// TwinCAT 3 PLC project SolidAttenuatorPLC
// ProgramVersion: 3.1.4022.7
// libraries:
//   lcls-twincat-motion, * (SLAC)
//   Tc2_Standard, * (Beckhoff Automation GmbH)
//   Tc2_System, * (Beckhoff Automation GmbH)
//   Tc3_Module, * (Beckhoff Automation GmbH)
//   VisuDialogs, * (System)
//   LCLS General,0.0.0,SLAC
//   VisuSymbols,3.5.10.0,System
// project tree:
//   DUTs/ DUT_MotionStage_Extras.TcDUT, ENUM_SXR_SATT_Position.TcDUT
//   / GlobalTextList.TcGTLO, PlcTask.TcTTO, VISU_TASK.TcTTO
//   GVLs/ Main.TcGVL
//   POUs/ FB_SXR_SATT_PositionState.TcPOU, FB_SXR_SATT_Stage.TcPOU, PRG_1_PlcTask.TcPOU, PRG_2_AT1K4.TcPOU
//   VISUs/ AT2K2_4022.TcVIS, VisualizationManager.TcVMO (not stored), VISU_MotionStage_4022.TcVIS, VISU_RTDs_4022.TcVIS
// real-time tasks:
//   TASK PlcTask: cycle T#10ms, priority 20, ADS port 350
//   TASK VISU_TASK: cycle T#200000us, priority 30, ADS port 351
// motion (NC):
//   TASK NC-Task 1 SAF: cycle T#2ms, priority 4, ADS port 501
//   TASK NC-Task 1 SVB: cycle T#10ms, priority 8, ADS port 511
//   AXIS AT1K4-M1 (id 1)
//     Dynamic: AccelerationMaximum=400, DecelerationMaximum=400, Acceleration=160, Deceleration=160, Jerk=80, DelayTime=0.008
//     Velo: Maximum=80
//     OtherSettings: AllowMotionCmdToSlave=true
//     encoder EncType=29
//       EncPara: ScaleFactorNumerator=5e-05, MaxCount=#xffffffff
//         SoftEndMinControl: Enable=true, Range=16.5
//         SoftEndMaxControl: Enable=true, Range=152.5
//         Inc: RefSoftSyncMask=#x0000ffff
//     drive DrvType=24
//       Analog: VeloReferenz=40, ScaleFactorActTorque=0.1
//       TimeComp: TaskDelayCycles=1
//     controller CtrType=2
//       CtrPara: PriorControlFactor=1
//         PosDiffControl: Range=0.2
//         PID: PosKp=20, PosExtKp=1, PosExtVelo=0.1
//         Observer: BandWidth=20
//   AXIS AT1K4-M2 (id 2)
//     Dynamic: AccelerationMaximum=400, DecelerationMaximum=400, Acceleration=160, Deceleration=160, Jerk=80, DelayTime=0.008
//     Velo: Maximum=80
//     OtherSettings: AllowMotionCmdToSlave=true
//     encoder EncType=29
//       EncPara: ScaleFactorNumerator=5e-05, MaxCount=#xffffffff, ReferenceSystem=1
//         SoftEndMinControl: Enable=true, Range=16.5
//         SoftEndMaxControl: Enable=true, Range=152.5
//         Inc: RefSoftSyncMask=#x0000ffff
//     drive DrvType=24
//       Analog: VeloReferenz=40, ScaleFactorActTorque=0.1
//       TimeComp: TaskDelayCycles=1
//     controller CtrType=2
//       CtrPara: PriorControlFactor=1
//         PosDiffControl: Range=0.2
//         PID: PosKp=20, PosExtKp=1, PosExtVelo=0.1
//         Observer: BandWidth=20
//   AXIS AT1K4-M3 (id 3)
//     Dynamic: AccelerationMaximum=400, DecelerationMaximum=400, Acceleration=160, Deceleration=160, Jerk=80, DelayTime=0.008
//     Velo: Maximum=80
//     OtherSettings: AllowMotionCmdToSlave=true
//     encoder EncType=29
//       EncPara: ScaleFactorNumerator=5e-05, MaxCount=#xffffffff, ReferenceSystem=1
//         SoftEndMinControl: Enable=true, Range=16.5
//         SoftEndMaxControl: Enable=true, Range=152.5
//         Inc: RefSoftSyncMask=#x0000ffff
//     drive DrvType=24
//       Analog: VeloReferenz=40, ScaleFactorActTorque=0.1
//       TimeComp: TaskDelayCycles=1
//     controller CtrType=2
//       CtrPara: PriorControlFactor=1
//         PosDiffControl: Range=0.2
//         PID: PosKp=20, PosExtKp=1, PosExtVelo=0.1
//         Observer: BandWidth=20
//   AXIS AT1K4-M4 (id 4)
//     Dynamic: AccelerationMaximum=400, DecelerationMaximum=400, Acceleration=160, Deceleration=160, Jerk=80, DelayTime=0.008
//     Velo: Maximum=80
//     OtherSettings: AllowMotionCmdToSlave=true
//     encoder EncType=29
//       EncPara: ScaleFactorNumerator=5e-05, MaxCount=#xffffffff, ReferenceSystem=1
//         SoftEndMinControl: Enable=true, Range=16.5
//         SoftEndMaxControl: Enable=true, Range=152.5
//         Inc: RefSoftSyncMask=#x0000ffff
//     drive DrvType=24
//       Analog: VeloReferenz=40, ScaleFactorActTorque=0.1
//       TimeComp: TaskDelayCycles=1
//     controller CtrType=2
//       CtrPara: PriorControlFactor=1
//         PosDiffControl: Range=0.2
//         PID: PosKp=20, PosExtKp=1, PosExtVelo=0.1
//         Observer: BandWidth=20
// I/O:
//   DEVICE Device 1 (EtherCAT), AmsNetId 172.21.148.185.2.1
//     Term 1 (EK1200) [EK1200-5000 EtherCAT Power supply (2A E-Bus)]
//       Term 14 (EL6695) [EL6695 EtherCAT Bridge terminal (Primary)]
//       Term 15 (EK1110) [EK1110 EtherCAT extension]
//     Term 16 (EK1100) [EK1100 EtherCAT Coupler (2A E-Bus)]
//       AT1K4-EL7047-01
//       AT1K4-EL7047-02 [EL7047 1Ch. Stepper motor output stage (50V, 5A)]
//       AT1K4-EL7047-03
//       AT1K4-EL7047-04
//       AT1K4-EL5042-01
//       AT1K4-EL5042-02
//       AT1K4-EL3202-01 [EL3202-0020 2Ch. Ana. Input PT100 (RTD), High Precision, calibrated]
//       AT1K4-EL3202-02 [EL3202-0020 2Ch. Ana. Input PT100 (RTD), High Precision, calibrated]
//       AT1K4-EL3202-03 [EL3202-0020 2Ch. Ana. Input PT100 (RTD), High Precision, calibrated]
//       AT1K4-EL3202-04 [EL3202-0020 2Ch. Ana. Input PT100 (RTD), High Precision, calibrated]
//       Term 12 (EL9011)
//   DEVICE Device 2 (EtherCAT Automation Protocol) (disabled), AmsNetId 172.21.148.185.3.1
//   DEVICE Device 5 (RT-Ethernet Protocol) (disabled), AmsNetId 172.21.148.185.6.1
//   DEVICE Device 4 (USB) (disabled)
//   DEVICE Device 6 (NOV-DP-RAM)
// variable links:
//   (this object) <-> Device 1 (EtherCAT)/Term 16 (EK1100)/AT1K4-EL5042-01
//     Enc/Inputs/In/nComState @bit 1 <-> WcState/InputToggle
//     Enc/Inputs/In/nComState <-> WcState/WcState
//     Enc/Inputs/In/nDataIn1 <-> FB Inputs Channel 1/Position
//     Enc/Inputs/In/nDataIn1 <-> FB Inputs Channel 2/Position
//     Enc/Inputs/In/nState1 @bit 12 <-> FB Inputs Channel 1/Status/Diag
//     Enc/Inputs/In/nState1 @bit 12 <-> FB Inputs Channel 2/Status/Diag
//     Enc/Inputs/In/nState1 @bit 1 <-> FB Inputs Channel 1/Status/Error
//     Enc/Inputs/In/nState1 @bit 1 <-> FB Inputs Channel 2/Status/Error
//     Enc/Inputs/In/nState1 @bit 14 <-> FB Inputs Channel 1/Status/Input cycle counter
//     Enc/Inputs/In/nState1 @bit 14 <-> FB Inputs Channel 2/Status/Input cycle counter
//     Enc/Inputs/In/nState1 @bit 2 <-> FB Inputs Channel 1/Status/Ready
//     Enc/Inputs/In/nState1 @bit 2 <-> FB Inputs Channel 2/Status/Ready
//     Enc/Inputs/In/nState1 @bit 13 <-> FB Inputs Channel 1/Status/TxPDO State
//     Enc/Inputs/In/nState1 @bit 13 <-> FB Inputs Channel 2/Status/TxPDO State
//     Enc/Inputs/In/nState1 <-> FB Inputs Channel 1/Status/Warning
//     Enc/Inputs/In/nState1 <-> FB Inputs Channel 2/Status/Warning
//   (this object) <-> Device 1 (EtherCAT)/Term 16 (EK1100)/AT1K4-EL7047-01
//     Drive/Inputs/In/nState1 @bit 3 <-> STM Status/Status/Error
//     Drive/Inputs/In/nState1 @bit 7 <-> STM Status/Status/Motor stall
//     Drive/Inputs/In/nState1 @bit 5 <-> STM Status/Status/Moving negative
//     Drive/Inputs/In/nState1 @bit 4 <-> STM Status/Status/Moving positive
//     Drive/Inputs/In/nState1 @bit 1 <-> STM Status/Status/Ready
//     Drive/Inputs/In/nState1 <-> STM Status/Status/Ready to enable
//     Drive/Inputs/In/nState1 @bit 6 <-> STM Status/Status/Torque reduced
//     Drive/Inputs/In/nState1 @bit 2 <-> STM Status/Status/Warning
//     Drive/Inputs/In/nState2 @bit 3 <-> STM Status/Status/Digital input 1
//     Drive/Inputs/In/nState2 @bit 4 <-> STM Status/Status/Digital input 2
//     Drive/Inputs/In/nState2 @bit 5 <-> STM Status/Status/Sync error
//     Drive/Inputs/In/nState2 @bit 7 <-> STM Status/Status/TxPDO Toggle
//     Drive/Inputs/In/nState4 @bit 1 <-> WcState/InputToggle
//     Drive/Inputs/In/nState4 <-> WcState/WcState
//     Drive/Outputs/Out/nCtrl1 <-> STM Control/Control/Enable
//     Drive/Outputs/Out/nCtrl1 @bit 2 <-> STM Control/Control/Reduce torque
//     Drive/Outputs/Out/nCtrl1 @bit 1 <-> STM Control/Control/Reset
//     Drive/Outputs/Out/nCtrl2 @bit 3 <-> STM Control/Control/Digital output 1
//     Drive/Outputs/Out/nDataOut2[0] <-> STM Velocity/Velocity
//   (this object) <-> Device 1 (EtherCAT)/Term 16 (EK1100)/AT1K4-EL7047-02
//     Drive/Inputs/In/nState1 @bit 3 <-> STM Status/Status/Error
//     Drive/Inputs/In/nState1 @bit 7 <-> STM Status/Status/Motor stall
//     Drive/Inputs/In/nState1 @bit 5 <-> STM Status/Status/Moving negative
//     Drive/Inputs/In/nState1 @bit 4 <-> STM Status/Status/Moving positive
//     Drive/Inputs/In/nState1 @bit 1 <-> STM Status/Status/Ready
//     Drive/Inputs/In/nState1 <-> STM Status/Status/Ready to enable
//     Drive/Inputs/In/nState1 @bit 6 <-> STM Status/Status/Torque reduced
//     Drive/Inputs/In/nState1 @bit 2 <-> STM Status/Status/Warning
//     Drive/Inputs/In/nState2 @bit 3 <-> STM Status/Status/Digital input 1
//     Drive/Inputs/In/nState2 @bit 4 <-> STM Status/Status/Digital input 2
//     Drive/Inputs/In/nState2 @bit 5 <-> STM Status/Status/Sync error
//     Drive/Inputs/In/nState2 @bit 7 <-> STM Status/Status/TxPDO Toggle
//     Drive/Inputs/In/nState4 @bit 1 <-> WcState/InputToggle
//     Drive/Inputs/In/nState4 <-> WcState/WcState
//     Drive/Outputs/Out/nCtrl1 <-> STM Control/Control/Enable
//     Drive/Outputs/Out/nCtrl1 @bit 2 <-> STM Control/Control/Reduce torque
//     Drive/Outputs/Out/nCtrl1 @bit 1 <-> STM Control/Control/Reset
//     Drive/Outputs/Out/nCtrl2 @bit 3 <-> STM Control/Control/Digital output 1
//     Drive/Outputs/Out/nDataOut2[0] <-> STM Velocity/Velocity
//   (this object) <-> Device 1 (EtherCAT)/Term 16 (EK1100)/AT1K4-EL5042-02
//     Enc/Inputs/In/nComState @bit 1 <-> WcState/InputToggle
//     Enc/Inputs/In/nComState <-> WcState/WcState
//     Enc/Inputs/In/nDataIn1 <-> FB Inputs Channel 1/Position
//     Enc/Inputs/In/nDataIn1 <-> FB Inputs Channel 2/Position
//     Enc/Inputs/In/nState1 @bit 12 <-> FB Inputs Channel 1/Status/Diag
//     Enc/Inputs/In/nState1 @bit 12 <-> FB Inputs Channel 2/Status/Diag
//     Enc/Inputs/In/nState1 @bit 1 <-> FB Inputs Channel 1/Status/Error
//     Enc/Inputs/In/nState1 @bit 1 <-> FB Inputs Channel 2/Status/Error
//     Enc/Inputs/In/nState1 @bit 14 <-> FB Inputs Channel 1/Status/Input cycle counter
//     Enc/Inputs/In/nState1 @bit 14 <-> FB Inputs Channel 2/Status/Input cycle counter
//     Enc/Inputs/In/nState1 @bit 2 <-> FB Inputs Channel 1/Status/Ready
//     Enc/Inputs/In/nState1 @bit 2 <-> FB Inputs Channel 2/Status/Ready
//     Enc/Inputs/In/nState1 @bit 13 <-> FB Inputs Channel 1/Status/TxPDO State
//     Enc/Inputs/In/nState1 @bit 13 <-> FB Inputs Channel 2/Status/TxPDO State
//     Enc/Inputs/In/nState1 <-> FB Inputs Channel 1/Status/Warning
//     Enc/Inputs/In/nState1 <-> FB Inputs Channel 2/Status/Warning
//   (this object) <-> Device 1 (EtherCAT)/Term 16 (EK1100)/AT1K4-EL7047-03
//     Drive/Inputs/In/nState1 @bit 3 <-> STM Status/Status/Error
//     Drive/Inputs/In/nState1 @bit 7 <-> STM Status/Status/Motor stall
//     Drive/Inputs/In/nState1 @bit 5 <-> STM Status/Status/Moving negative
//     Drive/Inputs/In/nState1 @bit 4 <-> STM Status/Status/Moving positive
//     Drive/Inputs/In/nState1 @bit 1 <-> STM Status/Status/Ready
//     Drive/Inputs/In/nState1 <-> STM Status/Status/Ready to enable
//     Drive/Inputs/In/nState1 @bit 6 <-> STM Status/Status/Torque reduced
//     Drive/Inputs/In/nState1 @bit 2 <-> STM Status/Status/Warning
//     Drive/Inputs/In/nState2 @bit 3 <-> STM Status/Status/Digital input 1
//     Drive/Inputs/In/nState2 @bit 4 <-> STM Status/Status/Digital input 2
//     Drive/Inputs/In/nState2 @bit 5 <-> STM Status/Status/Sync error
//     Drive/Inputs/In/nState2 @bit 7 <-> STM Status/Status/TxPDO Toggle
//     Drive/Inputs/In/nState4 @bit 1 <-> WcState/InputToggle
//     Drive/Inputs/In/nState4 <-> WcState/WcState
//     Drive/Outputs/Out/nCtrl1 <-> STM Control/Control/Enable
//     Drive/Outputs/Out/nCtrl1 @bit 2 <-> STM Control/Control/Reduce torque
//     Drive/Outputs/Out/nCtrl1 @bit 1 <-> STM Control/Control/Reset
//     Drive/Outputs/Out/nCtrl2 @bit 3 <-> STM Control/Control/Digital output 1
//     Drive/Outputs/Out/nDataOut2[0] <-> STM Velocity/Velocity
//   (this object) <-> Device 1 (EtherCAT)/Term 16 (EK1100)/AT1K4-EL7047-04
//     Drive/Inputs/In/nState1 @bit 3 <-> STM Status/Status/Error
//     Drive/Inputs/In/nState1 @bit 7 <-> STM Status/Status/Motor stall
//     Drive/Inputs/In/nState1 @bit 5 <-> STM Status/Status/Moving negative
//     Drive/Inputs/In/nState1 @bit 4 <-> STM Status/Status/Moving positive
//     Drive/Inputs/In/nState1 @bit 1 <-> STM Status/Status/Ready
//     Drive/Inputs/In/nState1 <-> STM Status/Status/Ready to enable
//     Drive/Inputs/In/nState1 @bit 6 <-> STM Status/Status/Torque reduced
//     Drive/Inputs/In/nState1 @bit 2 <-> STM Status/Status/Warning
//     Drive/Inputs/In/nState2 @bit 3 <-> STM Status/Status/Digital input 1
//     Drive/Inputs/In/nState2 @bit 4 <-> STM Status/Status/Digital input 2
//     Drive/Inputs/In/nState2 @bit 5 <-> STM Status/Status/Sync error
//     Drive/Inputs/In/nState2 @bit 7 <-> STM Status/Status/TxPDO Toggle
//     Drive/Inputs/In/nState4 @bit 1 <-> WcState/InputToggle
//     Drive/Inputs/In/nState4 <-> WcState/WcState
//     Drive/Outputs/Out/nCtrl1 <-> STM Control/Control/Enable
//     Drive/Outputs/Out/nCtrl1 @bit 2 <-> STM Control/Control/Reduce torque
//     Drive/Outputs/Out/nCtrl1 @bit 1 <-> STM Control/Control/Reset
//     Drive/Outputs/Out/nCtrl2 @bit 3 <-> STM Control/Control/Digital output 1
//     Drive/Outputs/Out/nDataOut2[0] <-> STM Velocity/Velocity
//   SolidAttenuatorPLC Instance <-> Device 1 (EtherCAT)/Term 16 (EK1100)/AT1K4-EL3202-01
//     PlcTask Inputs/PRG_2_AT1K4.fbStage1.fbRTD_1.bError <-> RTD Inputs Channel 1/Status/Error
//     PlcTask Inputs/PRG_2_AT1K4.fbStage1.fbRTD_2.bError <-> RTD Inputs Channel 2/Status/Error
//     PlcTask Inputs/PRG_2_AT1K4.fbStage1.fbRTD_1.bOverrange <-> RTD Inputs Channel 1/Status/Overrange
//     PlcTask Inputs/PRG_2_AT1K4.fbStage1.fbRTD_2.bOverrange <-> RTD Inputs Channel 2/Status/Overrange
//     PlcTask Inputs/PRG_2_AT1K4.fbStage1.fbRTD_1.bUnderrange <-> RTD Inputs Channel 1/Status/Underrange
//     PlcTask Inputs/PRG_2_AT1K4.fbStage1.fbRTD_2.bUnderrange <-> RTD Inputs Channel 2/Status/Underrange
//     PlcTask Inputs/PRG_2_AT1K4.fbStage1.fbRTD_1.iRaw <-> RTD Inputs Channel 1/Value
//     PlcTask Inputs/PRG_2_AT1K4.fbStage1.fbRTD_2.iRaw <-> RTD Inputs Channel 2/Value
//   SolidAttenuatorPLC Instance <-> Device 1 (EtherCAT)/Term 16 (EK1100)/AT1K4-EL3202-02
//     PlcTask Inputs/PRG_2_AT1K4.fbStage2.fbRTD_1.bError <-> RTD Inputs Channel 1/Status/Error
//     PlcTask Inputs/PRG_2_AT1K4.fbStage2.fbRTD_2.bError <-> RTD Inputs Channel 2/Status/Error
//     PlcTask Inputs/PRG_2_AT1K4.fbStage2.fbRTD_1.bOverrange <-> RTD Inputs Channel 1/Status/Overrange
//     PlcTask Inputs/PRG_2_AT1K4.fbStage2.fbRTD_2.bOverrange <-> RTD Inputs Channel 2/Status/Overrange
//     PlcTask Inputs/PRG_2_AT1K4.fbStage2.fbRTD_1.bUnderrange <-> RTD Inputs Channel 1/Status/Underrange
//     PlcTask Inputs/PRG_2_AT1K4.fbStage2.fbRTD_2.bUnderrange <-> RTD Inputs Channel 2/Status/Underrange
//     PlcTask Inputs/PRG_2_AT1K4.fbStage2.fbRTD_1.iRaw <-> RTD Inputs Channel 1/Value
//     PlcTask Inputs/PRG_2_AT1K4.fbStage2.fbRTD_2.iRaw <-> RTD Inputs Channel 2/Value
//   SolidAttenuatorPLC Instance <-> Device 1 (EtherCAT)/Term 16 (EK1100)/AT1K4-EL3202-03
//     PlcTask Inputs/PRG_2_AT1K4.fbStage3.fbRTD_1.bError <-> RTD Inputs Channel 1/Status/Error
//     PlcTask Inputs/PRG_2_AT1K4.fbStage3.fbRTD_2.bError <-> RTD Inputs Channel 2/Status/Error
//     PlcTask Inputs/PRG_2_AT1K4.fbStage3.fbRTD_1.bOverrange <-> RTD Inputs Channel 1/Status/Overrange
//     PlcTask Inputs/PRG_2_AT1K4.fbStage3.fbRTD_2.bOverrange <-> RTD Inputs Channel 2/Status/Overrange
//     PlcTask Inputs/PRG_2_AT1K4.fbStage3.fbRTD_1.bUnderrange <-> RTD Inputs Channel 1/Status/Underrange
//     PlcTask Inputs/PRG_2_AT1K4.fbStage3.fbRTD_2.bUnderrange <-> RTD Inputs Channel 2/Status/Underrange
//     PlcTask Inputs/PRG_2_AT1K4.fbStage3.fbRTD_1.iRaw <-> RTD Inputs Channel 1/Value
//     PlcTask Inputs/PRG_2_AT1K4.fbStage3.fbRTD_2.iRaw <-> RTD Inputs Channel 2/Value
//   SolidAttenuatorPLC Instance <-> Device 1 (EtherCAT)/Term 16 (EK1100)/AT1K4-EL3202-04
//     PlcTask Inputs/PRG_2_AT1K4.fbStage4.fbRTD_1.bError <-> RTD Inputs Channel 1/Status/Error
//     PlcTask Inputs/PRG_2_AT1K4.fbStage4.fbRTD_2.bError <-> RTD Inputs Channel 2/Status/Error
//     PlcTask Inputs/PRG_2_AT1K4.fbStage4.fbRTD_1.bOverrange <-> RTD Inputs Channel 1/Status/Overrange
//     PlcTask Inputs/PRG_2_AT1K4.fbStage4.fbRTD_2.bOverrange <-> RTD Inputs Channel 2/Status/Overrange
//     PlcTask Inputs/PRG_2_AT1K4.fbStage4.fbRTD_1.bUnderrange <-> RTD Inputs Channel 1/Status/Underrange
//     PlcTask Inputs/PRG_2_AT1K4.fbStage4.fbRTD_2.bUnderrange <-> RTD Inputs Channel 2/Status/Underrange
//     PlcTask Inputs/PRG_2_AT1K4.fbStage4.fbRTD_1.iRaw <-> RTD Inputs Channel 1/Value
//     PlcTask Inputs/PRG_2_AT1K4.fbStage4.fbRTD_2.iRaw <-> RTD Inputs Channel 2/Value
//   SolidAttenuatorPLC Instance <-> Device 1 (EtherCAT)/Term 16 (EK1100)/AT1K4-EL5042-01
//     PlcTask Inputs/Main.M1.nRawEncoderULINT <-> FB Inputs Channel 1/Position
//     PlcTask Inputs/Main.M2.nRawEncoderULINT <-> FB Inputs Channel 2/Position
//   SolidAttenuatorPLC Instance <-> Device 1 (EtherCAT)/Term 16 (EK1100)/AT1K4-EL5042-02
//     PlcTask Inputs/Main.M3.nRawEncoderULINT <-> FB Inputs Channel 1/Position
//     PlcTask Inputs/Main.M4.nRawEncoderULINT <-> FB Inputs Channel 2/Position
//   SolidAttenuatorPLC Instance <-> Device 1 (EtherCAT)/Term 16 (EK1100)/AT1K4-EL7047-01
//     PlcTask Inputs/Main.M1.bLimitBackwardEnable <-> STM Status/Status/Digital input 2
//     PlcTask Inputs/Main.M1.bLimitForwardEnable <-> STM Status/Status/Digital input 1
//   SolidAttenuatorPLC Instance <-> Device 1 (EtherCAT)/Term 16 (EK1100)/AT1K4-EL7047-02
//     PlcTask Inputs/Main.M2.bLimitBackwardEnable <-> STM Status/Status/Digital input 2
//     PlcTask Inputs/Main.M2.bLimitForwardEnable <-> STM Status/Status/Digital input 1
//   SolidAttenuatorPLC Instance <-> Device 1 (EtherCAT)/Term 16 (EK1100)/AT1K4-EL7047-03
//     PlcTask Inputs/Main.M3.bLimitBackwardEnable <-> STM Status/Status/Digital input 2
//     PlcTask Inputs/Main.M3.bLimitForwardEnable <-> STM Status/Status/Digital input 1
//   SolidAttenuatorPLC Instance <-> Device 1 (EtherCAT)/Term 16 (EK1100)/AT1K4-EL7047-04
//     PlcTask Inputs/Main.M4.bLimitBackwardEnable <-> STM Status/Status/Digital input 2
//     PlcTask Inputs/Main.M4.bLimitForwardEnable <-> STM Status/Status/Digital input 1
//   SolidAttenuatorPLC Instance <-> NC-Task 1 SAF/Axes/AT1K4-M1
//     PlcTask Inputs/Main.M1.Axis.NcToPlc <-> Outputs/ToPlc
//     PlcTask Outputs/Main.M1.Axis.PlcToNc <-> Inputs/FromPlc
//   SolidAttenuatorPLC Instance <-> NC-Task 1 SAF/Axes/AT1K4-M2
//     PlcTask Inputs/Main.M2.Axis.NcToPlc <-> Outputs/ToPlc
//     PlcTask Outputs/Main.M2.Axis.PlcToNc <-> Inputs/FromPlc
//   SolidAttenuatorPLC Instance <-> NC-Task 1 SAF/Axes/AT1K4-M3
//     PlcTask Inputs/Main.M3.Axis.NcToPlc <-> Outputs/ToPlc
//     PlcTask Outputs/Main.M3.Axis.PlcToNc <-> Inputs/FromPlc
//   SolidAttenuatorPLC Instance <-> NC-Task 1 SAF/Axes/AT1K4-M4
//     PlcTask Inputs/Main.M4.Axis.NcToPlc <-> Outputs/ToPlc
//     PlcTask Outputs/Main.M4.Axis.PlcToNc <-> Inputs/FromPlc

CONFIGURATION SolidAttenuatorPLC
    RESOURCE PLC ON TwinCAT3
        TASK PlcTask(INTERVAL := T#10ms, PRIORITY := 20);
        TASK VISU_TASK(INTERVAL := T#200000us, PRIORITY := 30);
        PROGRAM PRG_1_PlcTask WITH PlcTask : PRG_1_PlcTask;
        PROGRAM VisuElems_Visu_Prg WITH VISU_TASK : VisuElems.Visu_Prg;
    END_RESOURCE
END_CONFIGURATION

// ---- DUTs/DUT_MotionStage_Extras.TcDUT
TYPE DUT_MotionStage_Extras :
STRUCT
    fVisuStep: LREAL;
    bVisuLowLim: BOOL;
    bVisuHighLim: BOOL;
END_STRUCT
END_TYPE

// ---- DUTs/ENUM_SXR_SATT_Position.TcDUT
{attribute 'qualified_only'}
TYPE ENUM_SXR_SATT_Position :
(
    UNKNOWN := 0, // UNKNOWN must be in slot 0 or the FB breaks
    OUT := 1, // OUT at slot 1 is a convention
    FILTER1 := 2,
    FILTER2 := 3,
    FILTER3 := 4,
    FILTER4 := 5
);
END_TYPE

// ---- GVLs/Main.TcGVL
{attribute 'qualified_only'}
VAR_GLOBAL
(*
    Only includes motor definitions for the IOC
    These are hard-coded to be Main.M#,
    but are very convenient to store in a GVL,
    hence the confusing namespace here

    This should be refactored once the IOC
    supports arbitrary ads paths for motors
*)
(*
    Four identical systems:
    Instr.		Area		ID#			Z (m)
    TMO			FEE			AT1K4-SOLID	748
    NEH 2.2		H2.2		AT1K2-SOLID	784
    NEH 2.2		H2.2		AT2K2-SOLID	788.8
    TXI			H1.1		AT1K3-SOLID	~763

*)
    {attribute 'pytmc' := 'pv: AT1K4:L2SI:MMS:01'}
    {attribute 'TcLinkTo' := '
        .bLimitForwardEnable  := TIIB[AT1K4-EL7047-01]^STM Status^Status^Digital input 1;
        .bLimitBackwardEnable := TIIB[AT1K4-EL7047-01]^STM Status^Status^Digital input 2;
        .nRawEncoderULINT     := TIIB[AT1K4-EL5042-01]^FB Inputs Channel 1^Position;
    '}
    M1: DUT_MotionStage := (sName := 'AT1K4:L2SI:MMS:01');

    {attribute 'pytmc' := 'pv: AT1K4:L2SI:MMS:02'}
    {attribute 'TcLinkTo' := '
        .bLimitForwardEnable  := TIIB[AT1K4-EL7047-02]^STM Status^Status^Digital input 1;
        .bLimitBackwardEnable := TIIB[AT1K4-EL7047-02]^STM Status^Status^Digital input 2;
        .nRawEncoderULINT     := TIIB[AT1K4-EL5042-01]^FB Inputs Channel 2^Position;
    '}
    M2: DUT_MotionStage := (sName := 'AT1K4:L2SI:MMS:02');

    {attribute 'pytmc' := 'pv: AT1K4:L2SI:MMS:03'}
    {attribute 'TcLinkTo' := '
        .bLimitForwardEnable  := TIIB[AT1K4-EL7047-03]^STM Status^Status^Digital input 1;
        .bLimitBackwardEnable := TIIB[AT1K4-EL7047-03]^STM Status^Status^Digital input 2;
        .nRawEncoderULINT     := TIIB[AT1K4-EL5042-02]^FB Inputs Channel 1^Position;
    '}
    M3: DUT_MotionStage := (sName := 'AT1K4:L2SI:MMS:03');

    {attribute 'pytmc' := 'pv: AT1K4:L2SI:MMS:04'}
    {attribute 'TcLinkTo' := '
        .bLimitForwardEnable  := TIIB[AT1K4-EL7047-04]^STM Status^Status^Digital input 1;
        .bLimitBackwardEnable := TIIB[AT1K4-EL7047-04]^STM Status^Status^Digital input 2;
        .nRawEncoderULINT     := TIIB[AT1K4-EL5042-02]^FB Inputs Channel 2^Position;
    '}
    M4: DUT_MotionStage := (sName := 'AT1K4:L2SI:MMS:04');

END_VAR

// ---- POUs/PRG_1_PlcTask.TcPOU

PROGRAM PRG_1_PlcTask
VAR
    fbLogHandler: FB_LogHandler;
END_VAR

fbLogHandler();

PRG_2_AT1K4();

END_PROGRAM

// ---- POUs/PRG_2_AT1K4.TcPOU
PROGRAM PRG_2_AT1K4
VAR
    (* TODO: use FALSE for simulation and production *)
    (* TODO: use TRUE when relying on visualization + actual hardware *)
    bDebug : BOOL := FALSE;

    nEnableMode : ENUM_StageEnableMode;

    {attribute 'pytmc' := 'pv: AT1K4:L2SI:MMS:01'}
    {attribute 'TcLinkTo' := '

        .fbRTD_1.iRaw := TIIB[AT1K4-EL3202-01]^RTD Inputs Channel 1^Value;
        .fbRTD_1.bError := TIIB[AT1K4-EL3202-01]^RTD Inputs Channel 1^Status^Error;
        .fbRTD_1.bUnderrange := TIIB[AT1K4-EL3202-01]^RTD Inputs Channel 1^Status^Underrange;
        .fbRTD_1.bOverrange := TIIB[AT1K4-EL3202-01]^RTD Inputs Channel 1^Status^Overrange;

        .fbRTD_2.iRaw := TIIB[AT1K4-EL3202-01]^RTD Inputs Channel 2^Value;
        .fbRTD_2.bError := TIIB[AT1K4-EL3202-01]^RTD Inputs Channel 2^Status^Error;
        .fbRTD_2.bUnderrange := TIIB[AT1K4-EL3202-01]^RTD Inputs Channel 2^Status^Underrange;
        .fbRTD_2.bOverrange := TIIB[AT1K4-EL3202-01]^RTD Inputs Channel 2^Status^Overrange;

    '}
    fbStage1: FB_SXR_SATT_Stage;

    {attribute 'pytmc' := 'pv: AT1K4:L2SI:MMS:02'}
    {attribute 'TcLinkTo' := '

        .fbRTD_1.iRaw := TIIB[AT1K4-EL3202-02]^RTD Inputs Channel 1^Value;
        .fbRTD_1.bError := TIIB[AT1K4-EL3202-02]^RTD Inputs Channel 1^Status^Error;
        .fbRTD_1.bUnderrange := TIIB[AT1K4-EL3202-02]^RTD Inputs Channel 1^Status^Underrange;
        .fbRTD_1.bOverrange := TIIB[AT1K4-EL3202-02]^RTD Inputs Channel 1^Status^Overrange;

        .fbRTD_2.iRaw := TIIB[AT1K4-EL3202-02]^RTD Inputs Channel 2^Value;
        .fbRTD_2.bError := TIIB[AT1K4-EL3202-02]^RTD Inputs Channel 2^Status^Error;
        .fbRTD_2.bUnderrange := TIIB[AT1K4-EL3202-02]^RTD Inputs Channel 2^Status^Underrange;
        .fbRTD_2.bOverrange := TIIB[AT1K4-EL3202-02]^RTD Inputs Channel 2^Status^Overrange;

    '}
    fbStage2: FB_SXR_SATT_Stage;

    {attribute 'pytmc' := 'pv: AT1K4:L2SI:MMS:03'}
    {attribute 'TcLinkTo' := '

        .fbRTD_1.iRaw := TIIB[AT1K4-EL3202-03]^RTD Inputs Channel 1^Value;
        .fbRTD_1.bError := TIIB[AT1K4-EL3202-03]^RTD Inputs Channel 1^Status^Error;
        .fbRTD_1.bUnderrange := TIIB[AT1K4-EL3202-03]^RTD Inputs Channel 1^Status^Underrange;
        .fbRTD_1.bOverrange := TIIB[AT1K4-EL3202-03]^RTD Inputs Channel 1^Status^Overrange;

        .fbRTD_2.iRaw := TIIB[AT1K4-EL3202-03]^RTD Inputs Channel 2^Value;
        .fbRTD_2.bError := TIIB[AT1K4-EL3202-03]^RTD Inputs Channel 2^Status^Error;
        .fbRTD_2.bUnderrange := TIIB[AT1K4-EL3202-03]^RTD Inputs Channel 2^Status^Underrange;
        .fbRTD_2.bOverrange := TIIB[AT1K4-EL3202-03]^RTD Inputs Channel 2^Status^Overrange;
    '}
    fbStage3: FB_SXR_SATT_Stage;

    {attribute 'pytmc' := 'pv: AT1K4:L2SI:MMS:04'}
    {attribute 'TcLinkTo' := '

        .fbRTD_1.iRaw := TIIB[AT1K4-EL3202-04]^RTD Inputs Channel 1^Value;
        .fbRTD_1.bError := TIIB[AT1K4-EL3202-04]^RTD Inputs Channel 1^Status^Error;
        .fbRTD_1.bUnderrange := TIIB[AT1K4-EL3202-04]^RTD Inputs Channel 1^Status^Underrange;
        .fbRTD_1.bOverrange := TIIB[AT1K4-EL3202-04]^RTD Inputs Channel 1^Status^Overrange;

        .fbRTD_2.iRaw := TIIB[AT1K4-EL3202-04]^RTD Inputs Channel 2^Value;
        .fbRTD_2.bError := TIIB[AT1K4-EL3202-04]^RTD Inputs Channel 2^Status^Error;
        .fbRTD_2.bUnderrange := TIIB[AT1K4-EL3202-04]^RTD Inputs Channel 2^Status^Underrange;
        .fbRTD_2.bOverrange := TIIB[AT1K4-EL3202-04]^RTD Inputs Channel 2^Status^Overrange;
    '}
    fbStage4: FB_SXR_SATT_Stage;

END_VAR

IF bDebug THEN
    // NEVER: checkouts with the TwinCAT NC GUI.
    nEnableMode := ENUM_StageEnableMode.NEVER;
ELSE
    // ALWAYS: want active position correction at all times
    nEnableMode := ENUM_StageEnableMode.ALWAYS;
END_IF

(* State setup - stage 1 *)
fbStage1.stOut.sName         := 'Out';
fbStage1.stOut.fPosition     := 50;
fbStage1.stOut.fDelta        := 100;
fbStage1.stOut.fVelocity     := 10;
fbStage1.stOut.bValid        := TRUE;
fbStage1.stOut.bMoveOk       := TRUE;

fbStage1.stFilter1.sName     := 'Filter 1';
fbStage1.stFilter1.fPosition := 500;
fbStage1.stFilter1.fDelta    := 0;
fbStage1.stFilter1.fVelocity := 10;
fbStage1.stFilter1.bValid    := FALSE;
fbStage1.stFilter1.bMoveOk   := FALSE;

fbStage1.stFilter2.sName     := 'Filter 2';
fbStage1.stFilter2.fPosition := 500;
fbStage1.stFilter2.fDelta    := 0;
fbStage1.stFilter2.fVelocity := 10;
fbStage1.stFilter2.bValid    := FALSE;
fbStage1.stFilter2.bMoveOk   := FALSE;

fbStage1.stFilter3.sName     := 'Filter 3';
fbStage1.stFilter3.fPosition := 500;
fbStage1.stFilter3.fDelta    := 0;
fbStage1.stFilter3.fVelocity := 10;
fbStage1.stFilter3.bValid    := FALSE;
fbStage1.stFilter3.bMoveOk   := FALSE;

fbStage1.stFilter4.sName     := 'Filter 4';
fbStage1.stFilter4.fPosition := 500;
fbStage1.stFilter4.fDelta    := 0;
fbStage1.stFilter4.fVelocity := 10;
fbStage1.stFilter4.bValid    := FALSE;
fbStage1.stFilter4.bMoveOk   := FALSE;

fbStage1(stAxis:=Main.M1, nEnableMode:=nEnableMode);

(* State setup - stage 2 *)
fbStage2.stOut.sName         := 'Out';
fbStage2.stOut.fPosition     := 50;
fbStage2.stOut.fDelta        := 100;
fbStage2.stOut.fVelocity     := 10;
fbStage2.stOut.bValid        := TRUE;
fbStage2.stOut.bMoveOk       := TRUE;

fbStage2.stFilter1.sName     := 'Filter 1';
fbStage2.stFilter1.fPosition := 500;
fbStage2.stFilter1.fDelta    := 0;
fbStage2.stFilter1.fVelocity := 10;
fbStage2.stFilter1.bValid    := FALSE;
fbStage2.stFilter1.bMoveOk   := FALSE;

fbStage2.stFilter2.sName     := 'Filter 2';
fbStage2.stFilter2.fPosition := 500;
fbStage2.stFilter2.fDelta    := 0;
fbStage2.stFilter2.fVelocity := 10;
fbStage2.stFilter2.bValid    := FALSE;
fbStage2.stFilter2.bMoveOk   := FALSE;

fbStage2.stFilter3.sName     := 'Filter 3';
fbStage2.stFilter3.fPosition := 500;
fbStage2.stFilter3.fDelta    := 0;
fbStage2.stFilter3.fVelocity := 10;
fbStage2.stFilter3.bValid    := FALSE;
fbStage2.stFilter3.bMoveOk   := FALSE;

fbStage2.stFilter4.sName     := 'Filter 4';
fbStage2.stFilter4.fPosition := 500;
fbStage2.stFilter4.fDelta    := 0;
fbStage2.stFilter4.fVelocity := 10;
fbStage2.stFilter4.bValid    := FALSE;
fbStage2.stFilter4.bMoveOk   := FALSE;

fbStage2(stAxis:=Main.M2, nEnableMode:=nEnableMode);

(* State setup - stage 3 *)
fbStage3.stOut.sName         := 'Out';
fbStage3.stOut.fPosition     := 50;
fbStage3.stOut.fDelta        := 100;
fbStage3.stOut.fVelocity     := 10;
fbStage3.stOut.bValid        := TRUE;
fbStage3.stOut.bMoveOk       := TRUE;

fbStage3.stFilter1.sName     := 'Filter 1';
fbStage3.stFilter1.fPosition := 500;
fbStage3.stFilter1.fDelta    := 0;
fbStage3.stFilter1.fVelocity := 10;
fbStage3.stFilter1.bValid    := FALSE;
fbStage3.stFilter1.bMoveOk   := FALSE;

fbStage3.stFilter2.sName     := 'Filter 2';
fbStage3.stFilter2.fPosition := 500;
fbStage3.stFilter2.fDelta    := 0;
fbStage3.stFilter2.fVelocity := 10;
fbStage3.stFilter2.bValid    := FALSE;
fbStage3.stFilter2.bMoveOk   := FALSE;

fbStage3.stFilter3.sName     := 'Filter 3';
fbStage3.stFilter3.fPosition := 500;
fbStage3.stFilter3.fDelta    := 0;
fbStage3.stFilter3.fVelocity := 10;
fbStage3.stFilter3.bValid    := FALSE;
fbStage3.stFilter3.bMoveOk   := FALSE;

fbStage3.stFilter4.sName     := 'Filter 4';
fbStage3.stFilter4.fPosition := 500;
fbStage3.stFilter4.fDelta    := 0;
fbStage3.stFilter4.fVelocity := 10;
fbStage3.stFilter4.bValid    := FALSE;
fbStage3.stFilter4.bMoveOk   := FALSE;

fbStage3(stAxis:=Main.M3, nEnableMode:=nEnableMode);

(* State setup - stage 4 *)
fbStage4.stOut.sName         := 'Out';
fbStage4.stOut.fPosition     := 50;
fbStage4.stOut.fDelta        := 100;
fbStage4.stOut.fVelocity     := 10;
fbStage4.stOut.bValid        := TRUE;
fbStage4.stOut.bMoveOk       := TRUE;

fbStage4.stFilter1.sName     := 'Filter 1';
fbStage4.stFilter1.fPosition := 500;
fbStage4.stFilter1.fDelta    := 0;
fbStage4.stFilter1.fVelocity := 10;
fbStage4.stFilter1.bValid    := FALSE;
fbStage4.stFilter1.bMoveOk   := FALSE;

fbStage4.stFilter2.sName     := 'Filter 2';
fbStage4.stFilter2.fPosition := 500;
fbStage4.stFilter2.fDelta    := 0;
fbStage4.stFilter2.fVelocity := 10;
fbStage4.stFilter2.bValid    := FALSE;
fbStage4.stFilter2.bMoveOk   := FALSE;

fbStage4.stFilter3.sName     := 'Filter 3';
fbStage4.stFilter3.fPosition := 500;
fbStage4.stFilter3.fDelta    := 0;
fbStage4.stFilter3.fVelocity := 10;
fbStage4.stFilter3.bValid    := FALSE;
fbStage4.stFilter3.bMoveOk   := FALSE;

fbStage4.stFilter4.sName     := 'Filter 4';
fbStage4.stFilter4.fPosition := 500;
fbStage4.stFilter4.fDelta    := 0;
fbStage4.stFilter4.fVelocity := 10;
fbStage4.stFilter4.bValid    := FALSE;
fbStage4.stFilter4.bMoveOk   := FALSE;

fbStage4(stAxis:=Main.M4, nEnableMode:=nEnableMode);

END_PROGRAM

// ---- POUs/FB_SXR_SATT_Stage.TcPOU
FUNCTION_BLOCK FB_SXR_SATT_Stage
VAR_IN_OUT
    stAxis : DUT_MotionStage;
END_VAR
VAR_INPUT
    nEnableMode : ENUM_StageEnableMode;

    stOut		: DUT_PositionState;
    stFilter1	: DUT_PositionState;
    stFilter2	: DUT_PositionState;
    stFilter3	: DUT_PositionState;
    stFilter4	: DUT_PositionState;
END_VAR
VAR_OUTPUT
    stExtra : DUT_MotionStage_Extras;
    fTemp1 : LREAL;
    fTemp2 : LREAL;
END_VAR
VAR
    // TODO: debug
    // fbMotion: FB_MotionStage;
    fbMotion: FB_MotionStageSim;

    {attribute 'pytmc' := '
         pv: STATE
    '}
    fbState 	: FB_SXR_SATT_PositionState;

    bInitialized: BOOL := FALSE;

    (* EL3202-0020: 0.01 °C per digit *)
    {attribute 'pytmc' := 'pv: RTD:1'}
    fbRTD_1: FB_TempSensor := ( fResolution:=0.01 );
    {attribute 'pytmc' := 'pv: RTD:2'}
    fbRTD_2: FB_TempSensor := ( fResolution:=0.01 );

END_VAR

IF NOT bInitialized THEN
    bInitialized := TRUE;

    (* Defaults for DUT_MotionStage *)
    stAxis.bHardwareEnable      := TRUE;
    stAxis.bLimitBackwardEnable := TRUE;
    stAxis.bLimitForwardEnable  := TRUE;
    stAxis.bPowerSelf           := TRUE;
    stAxis.nBrakeMode           := ENUM_StageBrakeMode.NO_BRAKE;
    stAxis.nHomingMode          := ENUM_EpicsHomeCmd.NONE;

    (* Defaults for visualization *)
    stExtra.fVisuStep			:= 0.1;

END_IF

fbRTD_1();
fTemp1 := fbRTD_1.fTemp;

fbRTD_2();
fTemp2 := fbRTD_2.fTemp;

stAxis.nEnableMode := nEnableMode;
fbMotion(stMotionStage:=stAxis);
fbState(
    bEnable:=TRUE,
    bReset:=FALSE,
    stMotionStage:=stAxis,
    stOut:=stOut,
    stFilter1:=stFilter1,
    stFilter2:=stFilter2,
    stFilter3:=stFilter3,
    stFilter4:=stFilter4
);

stExtra.bVisuHighLim := NOT stAxis.bAllForwardEnable;
stExtra.bVisuLowLim := NOT stAxis.bAllBackwardEnable;

END_FUNCTION_BLOCK

// ---- POUs/FB_SXR_SATT_PositionState.TcPOU
FUNCTION_BLOCK FB_SXR_SATT_PositionState EXTENDS FB_PositionStateBase
VAR_INPUT
     // The enum position to move to
     {attribute 'pytmc' := '
         pv: SET
         io: io
     '}
     enumSet: ENUM_SXR_SATT_Position;

    // NOTE: Do not pragma these, let it happen in the manager.
     // Information about the OUT position
     stOut		: DUT_PositionState;
     stFilter1	: DUT_PositionState;
     stFilter2	: DUT_PositionState;
     stFilter3	: DUT_PositionState;
     stFilter4	: DUT_PositionState;

END_VAR
VAR_OUTPUT
    // The enum state readback
    {attribute 'pytmc' := '
        pv: GET
        io: i
    '}
    enumGet: ENUM_SXR_SATT_Position;
END_VAR
VAR
    bInitialized: BOOL := FALSE;
END_VAR

IF NOT bInitialized THEN
    bInitialized := TRUE;

    arrStates[1] := stOut;
    arrStates[2] := stFilter1;
    arrStates[3] := stFilter2;
    arrStates[4] := stFilter3;
    arrStates[5] := stFilter4;

END_IF
setState := enumSet;
Exec();
enumGet := getState;
enumSet := setState;

END_FUNCTION_BLOCK

// ---- GlobalTextList.TcGTLO
TEXTLIST GlobalTextList
  468 = '%d'
  405 = '%f'
  425 = '%X'
  417 = '+'
  411 = '-'
  421 = '0 = Default Acceleration'
  423 = '0 = Default Deceleration'
  420 = 'Acceleration: %f'
  966 = 'Admin'
  17 = 'Axis 1'
  746 = 'Axis 2'
  124 = 'Axis 3'
  441 = 'Axis 4'
  650 = 'Axis X'
  588 = 'Channel 1: %.2f C'
  84 = 'Channel 1: %f C'
  809 = 'Channel 2: %.2f C'
  18 = 'Channel 2: %f C'
  415 = 'Clear'
  409 = 'Control'
  406 = 'Current Position'
  463 = 'Current Position (raw)'
  422 = 'Deceleration: %f'
  426 = 'Error Code'
  424 = 'Error:'
  413 = 'GO'
  414 = 'GO to set position'
  407 = 'High Limit Hit Indicator'
  404 = 'Low Limit Hit Indicator'
  408 = 'Moving:'
  823 = 'None'
  269 = 'Operator'
  721 = 'RTD1: %f C'
  433 = 'RTD2: %f C'
  878 = 'Service'
  410 = 'Set Position'
  418 = 'Settings'
  403 = 'Status'
  412 = 'Step Size'
  416 = 'STOP'
  917 = 'Temp 1: %f C'
  719 = 'Temp 2: %f C'
  647 = 'Temperature Sensors'
  865 = 'Thermocouple Readback'
  419 = 'Velocity: %f'
END_TEXTLIST

// ---- VISUs/AT2K2_4022.TcVIS
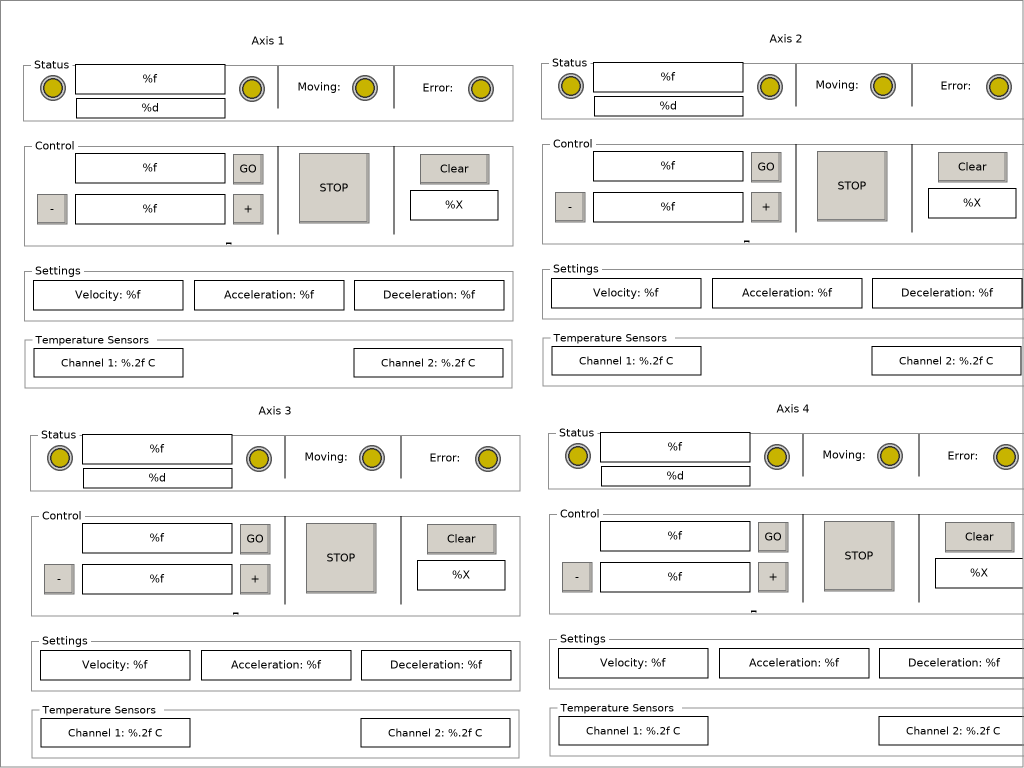
VISUALIZATION AT2K2_4022  // 1024x768
    Frame (8,40 520x300)
        shows VISU_MotionStage_4022(VisuMotionStage := Main.M1, Extras := PRG_2_AT1K4.fbStage1.stExtra)
    Label (193,26 150x30), "Axis 1"
    Frame (9,332 505x58)
        shows VISU_RTDs_4022(fTemp1 := PRG_2_AT1K4.fbStage1.fTemp1, fTemp2 := PRG_2_AT1K4.fbStage1.fTemp2)
    Frame (526,38 520x300)
        shows VISU_MotionStage_4022(VisuMotionStage := Main.M2, Extras := PRG_2_AT1K4.fbStage2.stExtra)
    Label (711,24 150x30), "Axis 2"
    Frame (527,330 505x58)
        shows VISU_RTDs_4022(fTemp1 := PRG_2_AT1K4.fbStage2.fTemp1, fTemp2 := PRG_2_AT1K4.fbStage2.fTemp2)
    Frame (15,410 520x300)
        shows VISU_MotionStage_4022(VisuMotionStage := Main.M3, Extras := PRG_2_AT1K4.fbStage3.stExtra)
    Label (200,396 150x30), "Axis 3"
    Frame (16,702 505x58)
        shows VISU_RTDs_4022(fTemp1 := PRG_2_AT1K4.fbStage3.fTemp1, fTemp2 := PRG_2_AT1K4.fbStage3.fTemp2)
    Frame (533,408 520x300)
        shows VISU_MotionStage_4022(VisuMotionStage := Main.M4, Extras := PRG_2_AT1K4.fbStage4.stExtra)
    Label (718,394 150x30), "Axis 4"
    Frame (534,700 505x58)
        shows VISU_RTDs_4022(fTemp1 := PRG_2_AT1K4.fbStage4.fTemp1, fTemp2 := PRG_2_AT1K4.fbStage4.fTemp2)
END_VISUALIZATION

// ---- VISUs/VISU_MotionStage_4022.TcVIS
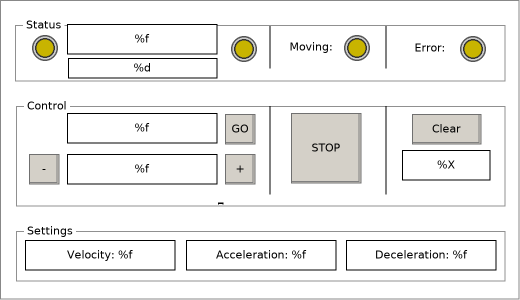
VISUALIZATION VISU_MotionStage_4022  // 520x300
VAR_IN_OUT
	VisuMotionStage: DUT_MotionStage;
	Extras: DUT_MotionStage_Extras;
END_VAR
    GroupBox (15,17 490x64), "Status"
        Lamp1 (15,16 30x30), tooltip "Low Limit Hit Indicator", variable: Extras.bVisuLowLim, style: Lamp-Lamp1-Yellow
        Rectangle (52,7 150x30), "%f", tooltip "Current Position", text variable: VisuMotionStage.stAxisStatus.fActPosition
        Lamp1 (214,17 30x30), tooltip "High Limit Hit Indicator", variable: Extras.bVisuHighLim, style: Lamp-Lamp1-Yellow
        Lamp1 (327,16 30x30), variable: VisuMotionStage.bBusy, style: Lamp-Lamp1-Yellow
        Label (262,15 68x30), "Moving:"
        Line (371,51) (371,9)
        Lamp1 (443,17 30x30), variable: VisuMotionStage.bError, style: Lamp-Lamp1-Yellow
    Rectangle (218,203 5x0)
    GroupBox (16,98 489x108), "Control"
        Rectangle (51,15 150x30), "%f", tooltip "Set Position", text variable: VisuMotionStage.fPosition
            OnMouseDown: write the text variable via Default
        Button (13,56 30x30), "-"
            OnMouseDown: execute {
                VisuMotionStage.nCommand := 3;
                VisuMotionStage.fPosition := VisuMotionStage.stAxisStatus.fActPosition - Extras.fVisuStep;
                VisuMotionStage.bExecute := TRUE;
            }
        Rectangle (51,56 150x30), "%f", tooltip "Step Size", text variable: Extras.fVisuStep
            OnMouseDown: write the text variable via Default
        Button (209,16 30x30), "GO", tooltip "GO to set position"
            OnMouseDown: execute { VisuMotionStage.nCommand := 3; VisuMotionStage.bExecute := TRUE; }
        Line (254,96) (254,8)
        Line (370,96) (370,8)
        Button (396,16 69x30), "Clear"
            tap VisuMotionStage.bReset
        Button (275,15 70x70), "STOP", tooltip "GO to set position"
            OnMouseDown: execute { VisuMotionStage.bExecute := FALSE; }
        Button (209,56 30x30), "+"
            OnMouseDown: execute {
                VisuMotionStage.nCommand := 3;
                VisuMotionStage.fPosition := VisuMotionStage.stAxisStatus.fActPosition + Extras.fVisuStep;
                VisuMotionStage.bExecute := TRUE;
            }
    GroupBox (16,223 489x58), "Settings"
        Rectangle (9,17 150x30), "Velocity: %f", text variable: VisuMotionStage.fVelocity
            OnMouseDown: write the text variable via Default
        Rectangle (170,17 150x30), "Acceleration: %f", tooltip "0 = Default Acceleration", text variable: VisuMotionStage.fAcceleration
            OnMouseDown: write the text variable via Default
        Rectangle (330,17 150x30), "Deceleration: %f", tooltip "0 = Default Deceleration", text variable: VisuMotionStage.fDeceleration
            OnMouseDown: write the text variable via Default
    Line (270,68) (270,26)
    Label (396,33 68x30), "Error:"
    Rectangle (402,150 88x30), "%X", tooltip "Error Code", text variable: VisuMotionStage.stAxisStatus.nErrorId
    Rectangle (68,58 149x20), "%d", tooltip "Current Position (raw)", text variable: VisuMotionStage.nRawEncoderULINT
END_VISUALIZATION

// ---- VISUs/VISU_RTDs_4022.TcVIS
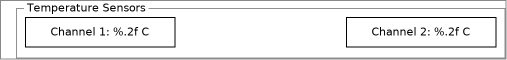
VISUALIZATION VISU_RTDs_4022  // 507x60
VAR_IN_OUT
	fTemp1 : LREAL;
	fTemp2 : LREAL;
END_VAR
    GroupBox (16,0 489x58), "Temperature Sensors"
        Rectangle (9,17 150x30), "Channel 1: %.2f C", text variable: fTemp1
            OnMouseDown: write the text variable via Default
        Rectangle (330,17 150x30), "Channel 2: %.2f C", tooltip "0 = Default Deceleration", text variable: fTemp2
            OnMouseDown: write the text variable via Default
END_VISUALIZATION
